// TIA Portal project "limit_switch" (V15)

(* hardware
DEVICE "S7-1200 station_1"  S7-1200 Station
   slot 0: "Rack_0"  S7-1200 Rack  Rack  V1.0
   slot 1: "PLC_1"  CPU 1212C AC/DC/Rly  6ES7 212-1BE40-0XB0  V4.0
*)

// ===== PLC "PLC_1"  CPU 1212C AC/DC/Rly =====

VAR_GLOBAL   // PLC tag table "Default tag table"
   "start" AT %I0.0 : Bool;
   "limt2" AT %I0.4 : Bool;
   "motor1" AT %Q0.0 : Bool;
   "limt3" AT %I0.5 : Bool;
   "motor2" AT %Q0.1 : Bool;
   "limt1" AT %I0.3 : Bool;
   "stop" AT %I0.2 : Bool;
   "mark1" AT %M0.0 : Bool;
   "markk" AT %M0.1 : Bool;
   "X" AT %M0.2 : Bool;
   "Tag_1" AT %M0.5 : Bool;
END_VAR

ORGANIZATION_BLOCK "Main"   // OB1, LAD, ProgramCycle
TITLE = "Main Program Sweep (Cycle)"
{ S7_Optimized_Access := 'TRUE' }
VERSION : 0.1
   VAR_INPUT
      Initial_Call : Bool;   // Initial call of this OB
      Remanence : Bool;   // =True, if remanent data are available
   END_VAR
BEGIN

REGION Network 1
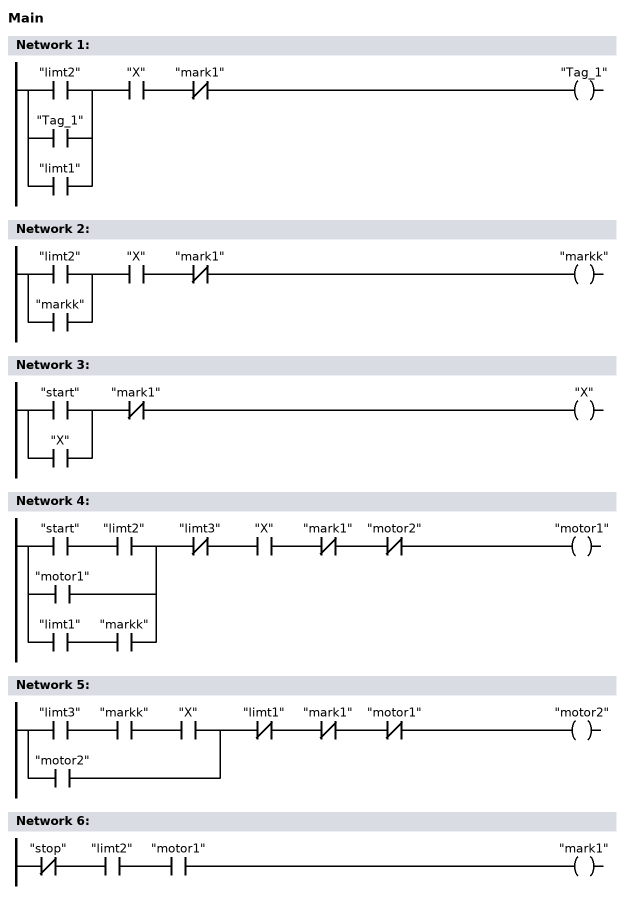
   RUNG wire#powerrail
      Contact( "limt2" )
      wire#w1
      Contact( "X" )
      I_Contact( "mark1" )
      Coil( "Tag_1" )
   END_RUNG
   RUNG wire#powerrail
      Contact( "Tag_1" )
   END_RUNG wire#w1
   RUNG wire#powerrail
      Contact( "limt1" )
   END_RUNG wire#w1
   // the same network as SCL:
   "Tag_1" := ("limt2" OR "Tag_1" OR "limt1") AND "X" AND NOT "mark1";
END_REGION

REGION Network 2
   RUNG wire#powerrail
      Contact( "limt2" )
      wire#w1
      Contact( "X" )
      I_Contact( "mark1" )
      Coil( "markk" )
   END_RUNG
   RUNG wire#powerrail
      Contact( "markk" )
   END_RUNG wire#w1
   // the same network as SCL:
   "markk" := ("limt2" OR "markk") AND "X" AND NOT "mark1";
END_REGION

REGION Network 3
   RUNG wire#powerrail
      Contact( "start" )
      wire#w1
      I_Contact( "mark1" )
      Coil( "X" )
   END_RUNG
   RUNG wire#powerrail
      Contact( "X" )
   END_RUNG wire#w1
   // the same network as SCL:
   "X" := ("start" OR "X") AND NOT "mark1";
END_REGION

REGION Network 4
   RUNG wire#powerrail
      Contact( "start" )
      Contact( "limt2" )
      wire#w1
      I_Contact( "limt3" )
      Contact( "X" )
      I_Contact( "mark1" )
      I_Contact( "motor2" )
      Coil( "motor1" )
   END_RUNG
   RUNG wire#powerrail
      Contact( "motor1" )
   END_RUNG wire#w1
   RUNG wire#powerrail
      Contact( "limt1" )
      Contact( "markk" )
   END_RUNG wire#w1
   // the same network as SCL:
   "motor1" := (("start" AND "limt2") OR "motor1" OR ("limt1" AND "markk")) AND NOT "limt3" AND "X" AND NOT "mark1" AND NOT "motor2";
END_REGION

REGION Network 5
   RUNG wire#powerrail
      Contact( "limt3" )
      Contact( "markk" )
      Contact( "X" )
      wire#w1
      I_Contact( "limt1" )
      I_Contact( "mark1" )
      I_Contact( "motor1" )
      Coil( "motor2" )
   END_RUNG
   RUNG wire#powerrail
      Contact( "motor2" )
   END_RUNG wire#w1
   // the same network as SCL:
   "motor2" := (("limt3" AND "markk" AND "X") OR "motor2") AND NOT "limt1" AND NOT "mark1" AND NOT "motor1";
END_REGION

REGION Network 6
   RUNG wire#powerrail
      I_Contact( "stop" )
      Contact( "limt2" )
      Contact( "motor1" )
      Coil( "mark1" )
   END_RUNG
   // the same network as SCL:
   "mark1" := NOT "stop" AND "limt2" AND "motor1";
END_REGION
END_ORGANIZATION_BLOCK